// TIA Portal V18 export
DATA_BLOCK "L1_ERP_packet"   // DB37
{ S7_Optimized_Access := 'TRUE' }
VERSION : 0.1
// stored: AutoNumber false, DBAccessibleFromOPCUA true, DBAccessibleFromWebserver true, IsOnlyStoredInLoadMemory false, IsRetainMemResEnabled false, IsWriteProtectedInAS false, MemoryReserve 100
   VAR
      eventlog_TEST : Bool;
      eventlog_PLC_PC { S7_SetPoint := 'True'} : Bool;   // Scrittura evento PLC
      eventlog_PC_PLC { S7_SetPoint := 'True'} : Bool;   // ack scrittura evento PC
      data : "LGasp_TypeERP_packet";   // dati pacco
   END_VAR
BEGIN
END_DATA_BLOCK
